// TIA Portal V17 export
// export: Created 2025-06-26T07:49:57.6660694Z, ExportSetting WithDefaults, DisplayName Totally Integrated Automation Portal, DisplayVersion V17 Update 8, DisplayName TIA Portal Openness, DisplayVersion V17 Update 8, DisplayName TIA Portal Version Control Interface, DisplayVersion V17, DisplayName STEP 7 Professional, DisplayVersion V17 Update 8, DisplayName STEP 7 Safety, DisplayVersion V17 Update 6, DisplayName WinCC Advanced, DisplayVersion V17 Update 8
TYPE "FluidData-STRUCT"
// stored: IsFailsafeCompliant false
   STRUCT
      "Name" : String;
      FluidTypeNumber : Int;
      SaturationCurve_Temperature_C : Array[0..40] of Real;
      SaturationCurve_Pressure_kPa : Array[0..40] of Real;
      DensityCurve_Pressure_kPa : Array[0..12] of Real;
      DensityCurveLiquide_Densety_kg_m3 : Array[0..12] of Real;
      DensityCurveVapor_Densety_kg_m3 : Array[0..12] of Real;
      DensityCurveVapor_SuperheatCorrection_a : Real;
      DensityCurveVapor_SuperheatCorrection_b : Real;
      EnthalpyMap_Superheat_C : Array[0..8] of Real;
      EnthalpyMap_Pressure_kPa : Array[0..11] of Real;
      EnthalpyMap_Enthalpy_kJ_kg : Array[0..11, 0..8] of Real;
      Limits { S7_SetPoint := 'True'} : "FluidBasedLimits-STRUCT";
      T_AdditionalSuperHeatEvaporator : Real;
      P_CriticalPoint : Real := 99999.9;
   END_STRUCT;
END_TYPE
